{attribute addProperty BoxType "EL6080-0000-0016"}
{attribute addProperty Id "StatusAT %I*Status_77B8DE54000InputsEMPTY_STRUCTURE000ControlAT %Q*Control_AB2F34C6000OutputsEMPTY_STRUCTURE000WcStateAT %I*WcState_98A4DF7520.250InfoDataAT %I*InfoData_BC63D37F80100"}
{attribute addProperty CRC "3689285382"}
{attribute addProperty SizeInBites "82"}
{attribute addProperty SizeInBytes "10.25"}
TYPE EL6080_AABC74D8 :
STRUCT
	{attribute addProperty Name "Status"}
	Status : Status_77B8DE54;
	{attribute addProperty Name "Inputs"}
	Inputs : EMPTY_STRUCTURE;
	{attribute addProperty Name "Control"}
	Control : Control_AB2F34C6;
	{attribute addProperty Name "Outputs"}
	Outputs : EMPTY_STRUCTURE;
	{attribute addProperty Name "WcState"}
	WcState : WcState_98A4DF75;
	{attribute addProperty Name "InfoData"}
	InfoData : InfoData_BC63D37F;
END_STRUCT
END_TYPE

(* stored: Version 1.2.0.0, ProductVersion 3.1.4024.9
   DUT EL6080_AABC74D8: Id {fcb96a11-9b98-47bd-b8e2-41a13344da5b} *)
